// TIA Portal V19 export
FUNCTION "A0303_Sollevamento_CALL" : Void   // FC148, LAD
// stored: SetENOAutomatically false
BEGIN

REGION Network 1: <<< LATO TESTA >>>
END_REGION

REGION Network 2: Data In - Ax
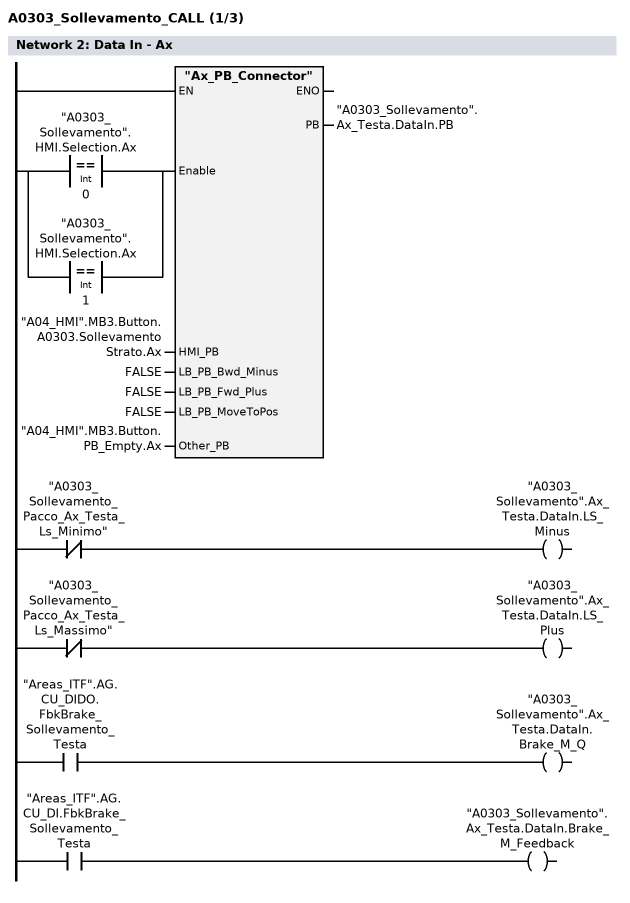
   RUNG wire#powerrail
      "Ax_PB_Connector"(Enable := wire#w1, HMI_PB := "A04_HMI".MB3.Button.A0303.SollevamentoStrato.Ax, LB_PB_Bwd_Minus := FALSE, LB_PB_Fwd_Plus := FALSE, LB_PB_MoveToPos := FALSE, Other_PB := "A04_HMI".MB3.Button.PB_Empty.Ax, PB => "A0303_Sollevamento".Ax_Testa.DataIn.PB)
   END_RUNG
   RUNG wire#powerrail
      { S7_Templates := "SrcType := Int" } EQ_Contact(in1 := "A0303_Sollevamento".HMI.Selection.Ax, in2 := 0)
   END_RUNG wire#w1
   RUNG wire#powerrail
      { S7_Templates := "SrcType := Int" } EQ_Contact(in1 := "A0303_Sollevamento".HMI.Selection.Ax, in2 := 1)
   END_RUNG wire#w1
   RUNG wire#powerrail
      I_Contact( "A0303_Sollevamento_Pacco_Ax_Testa_Ls_Minimo" )
      Coil( "A0303_Sollevamento".Ax_Testa.DataIn.LS_Minus )
   END_RUNG
   RUNG wire#powerrail
      I_Contact( "A0303_Sollevamento_Pacco_Ax_Testa_Ls_Massimo" )
      Coil( "A0303_Sollevamento".Ax_Testa.DataIn.LS_Plus )
   END_RUNG
   RUNG wire#powerrail
      Contact( "Areas_ITF".AG.CU_DIDO.FbkBrake_Sollevamento_Testa )
      Coil( "A0303_Sollevamento".Ax_Testa.DataIn.Brake_M_Q )
   END_RUNG
   RUNG wire#powerrail
      Contact( "Areas_ITF".AG.CU_DI.FbkBrake_Sollevamento_Testa )
      Coil( "A0303_Sollevamento".Ax_Testa.DataIn.Brake_M_Feedback )
   END_RUNG
   // the same network as SCL:
   "Ax_PB_Connector"(Enable := ("A0303_Sollevamento".HMI.Selection.Ax = 0) OR ("A0303_Sollevamento".HMI.Selection.Ax = 1),
                     HMI_PB := "A04_HMI".MB3.Button.A0303.SollevamentoStrato.Ax,
                     LB_PB_Bwd_Minus := FALSE,
                     LB_PB_Fwd_Plus := FALSE,
                     LB_PB_MoveToPos := FALSE,
                     Other_PB := "A04_HMI".MB3.Button.PB_Empty.Ax,
                     PB => "A0303_Sollevamento".Ax_Testa.DataIn.PB);
   "A0303_Sollevamento".Ax_Testa.DataIn.LS_Minus := NOT "A0303_Sollevamento_Pacco_Ax_Testa_Ls_Minimo";
   "A0303_Sollevamento".Ax_Testa.DataIn.LS_Plus := NOT "A0303_Sollevamento_Pacco_Ax_Testa_Ls_Massimo";
   "A0303_Sollevamento".Ax_Testa.DataIn.Brake_M_Q := "Areas_ITF".AG.CU_DIDO.FbkBrake_Sollevamento_Testa;
   "A0303_Sollevamento".Ax_Testa.DataIn.Brake_M_Feedback := "Areas_ITF".AG.CU_DI.FbkBrake_Sollevamento_Testa;
END_REGION

REGION Network 3: <<< LATO CODA >>>
END_REGION

REGION Network 4: Data In - Ax
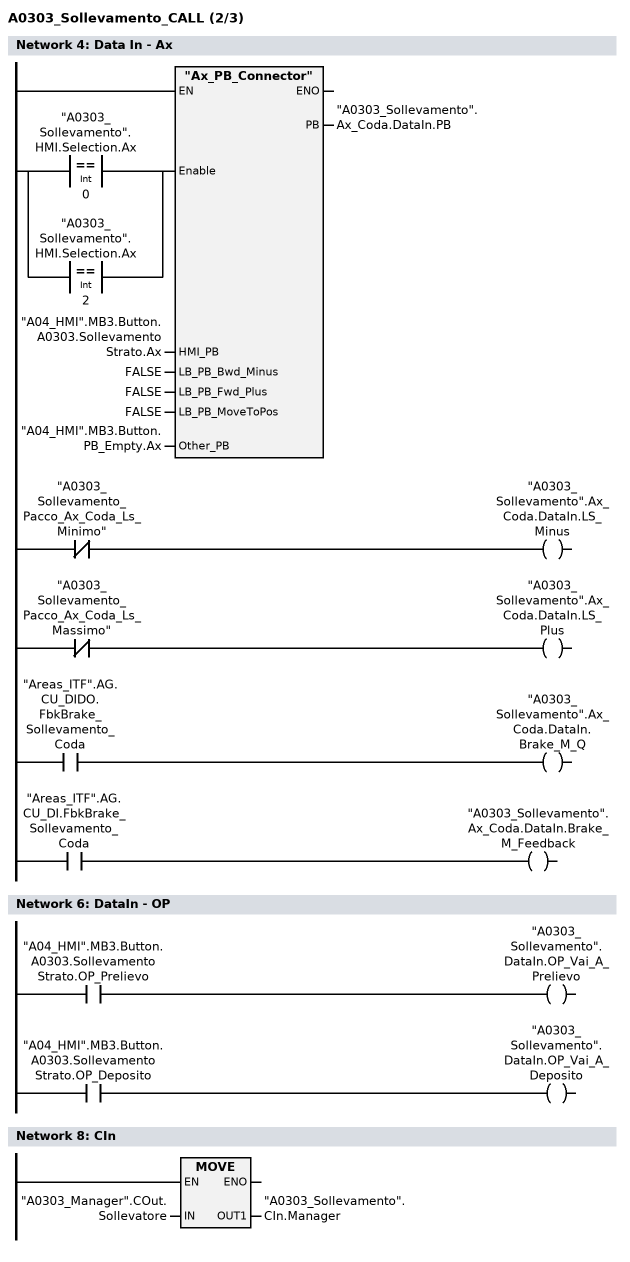
   RUNG wire#powerrail
      "Ax_PB_Connector"(Enable := wire#w1, HMI_PB := "A04_HMI".MB3.Button.A0303.SollevamentoStrato.Ax, LB_PB_Bwd_Minus := FALSE, LB_PB_Fwd_Plus := FALSE, LB_PB_MoveToPos := FALSE, Other_PB := "A04_HMI".MB3.Button.PB_Empty.Ax, PB => "A0303_Sollevamento".Ax_Coda.DataIn.PB)
   END_RUNG
   RUNG wire#powerrail
      { S7_Templates := "SrcType := Int" } EQ_Contact(in1 := "A0303_Sollevamento".HMI.Selection.Ax, in2 := 0)
   END_RUNG wire#w1
   RUNG wire#powerrail
      { S7_Templates := "SrcType := Int" } EQ_Contact(in1 := "A0303_Sollevamento".HMI.Selection.Ax, in2 := 2)
   END_RUNG wire#w1
   RUNG wire#powerrail
      I_Contact( "A0303_Sollevamento_Pacco_Ax_Coda_Ls_Minimo" )
      Coil( "A0303_Sollevamento".Ax_Coda.DataIn.LS_Minus )
   END_RUNG
   RUNG wire#powerrail
      I_Contact( "A0303_Sollevamento_Pacco_Ax_Coda_Ls_Massimo" )
      Coil( "A0303_Sollevamento".Ax_Coda.DataIn.LS_Plus )
   END_RUNG
   RUNG wire#powerrail
      Contact( "Areas_ITF".AG.CU_DIDO.FbkBrake_Sollevamento_Coda )
      Coil( "A0303_Sollevamento".Ax_Coda.DataIn.Brake_M_Q )
   END_RUNG
   RUNG wire#powerrail
      Contact( "Areas_ITF".AG.CU_DI.FbkBrake_Sollevamento_Coda )
      Coil( "A0303_Sollevamento".Ax_Coda.DataIn.Brake_M_Feedback )
   END_RUNG
   // the same network as SCL:
   "Ax_PB_Connector"(Enable := ("A0303_Sollevamento".HMI.Selection.Ax = 0) OR ("A0303_Sollevamento".HMI.Selection.Ax = 2),
                     HMI_PB := "A04_HMI".MB3.Button.A0303.SollevamentoStrato.Ax,
                     LB_PB_Bwd_Minus := FALSE,
                     LB_PB_Fwd_Plus := FALSE,
                     LB_PB_MoveToPos := FALSE,
                     Other_PB := "A04_HMI".MB3.Button.PB_Empty.Ax,
                     PB => "A0303_Sollevamento".Ax_Coda.DataIn.PB);
   "A0303_Sollevamento".Ax_Coda.DataIn.LS_Minus := NOT "A0303_Sollevamento_Pacco_Ax_Coda_Ls_Minimo";
   "A0303_Sollevamento".Ax_Coda.DataIn.LS_Plus := NOT "A0303_Sollevamento_Pacco_Ax_Coda_Ls_Massimo";
   "A0303_Sollevamento".Ax_Coda.DataIn.Brake_M_Q := "Areas_ITF".AG.CU_DIDO.FbkBrake_Sollevamento_Coda;
   "A0303_Sollevamento".Ax_Coda.DataIn.Brake_M_Feedback := "Areas_ITF".AG.CU_DI.FbkBrake_Sollevamento_Coda;
END_REGION

REGION Network 5: >
END_REGION

REGION Network 6: DataIn - OP
   RUNG wire#powerrail
      Contact( "A04_HMI".MB3.Button.A0303.SollevamentoStrato.OP_Prelievo )
      Coil( "A0303_Sollevamento".DataIn.OP_Vai_A_Prelievo )
   END_RUNG
   RUNG wire#powerrail
      Contact( "A04_HMI".MB3.Button.A0303.SollevamentoStrato.OP_Deposito )
      Coil( "A0303_Sollevamento".DataIn.OP_Vai_A_Deposito )
   END_RUNG
   // the same network as SCL:
   "A0303_Sollevamento".DataIn.OP_Vai_A_Prelievo := "A04_HMI".MB3.Button.A0303.SollevamentoStrato.OP_Prelievo;
   "A0303_Sollevamento".DataIn.OP_Vai_A_Deposito := "A04_HMI".MB3.Button.A0303.SollevamentoStrato.OP_Deposito;
END_REGION

REGION Network 7: >
END_REGION

REGION Network 8: CIn
   RUNG wire#powerrail
      Move(in := "A0303_Manager".COut.Sollevatore, out1 => "A0303_Sollevamento".CIn.Manager)
   END_RUNG
   // the same network as SCL:
   "A0303_Sollevamento".CIn.Manager := "A0303_Manager".COut.Sollevatore;
END_REGION

REGION Network 9: CIn Trasporto
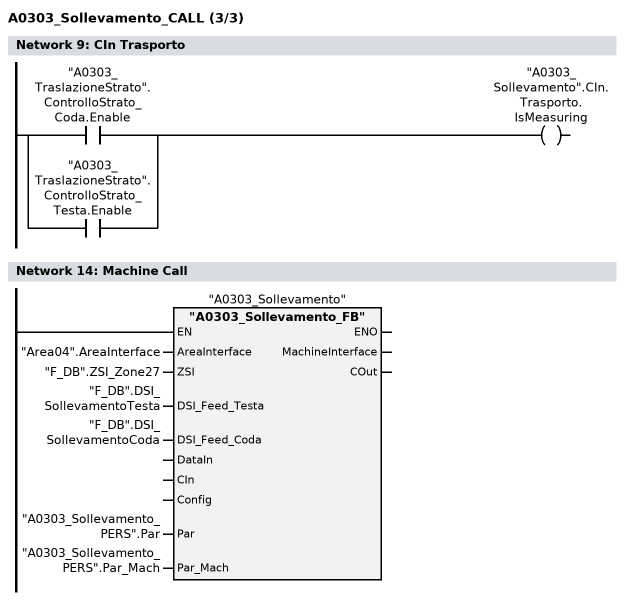
   RUNG wire#powerrail
      Contact( "A0303_TraslazioneStrato".ControlloStrato_Coda.Enable )
      wire#w1
      Coil( "A0303_Sollevamento".CIn.Trasporto.IsMeasuring )
   END_RUNG
   RUNG wire#powerrail
      Contact( "A0303_TraslazioneStrato".ControlloStrato_Testa.Enable )
   END_RUNG wire#w1
   // the same network as SCL:
   "A0303_Sollevamento".CIn.Trasporto.IsMeasuring := "A0303_TraslazioneStrato".ControlloStrato_Coda.Enable OR "A0303_TraslazioneStrato".ControlloStrato_Testa.Enable;
END_REGION

REGION Network 10: >
END_REGION

REGION Network 11 (SCL): Drive
   "A0303_Sollevamento".Ax_Testa.Drive.Infeed_ON := "Areas_ITF".AG.Infeed_Running;
   "A0303_Sollevamento".Ax_Testa.Drive.AccessPoint := "HW_Const_Values".CU8_PN_615A1_ModuleAccessPoint;
   "A0303_Sollevamento".Ax_Testa.Drive.AxisID := "CU8_ID_2_2390A1_1_2390M1";
   "A0303_Sollevamento".Ax_Testa.Drive.TokenChain := "TOKENCHAIN_CU8";

   "A0303_Sollevamento".Ax_Coda.Drive.Infeed_ON := "Areas_ITF".AG.Infeed_Running;
   "A0303_Sollevamento".Ax_Coda.Drive.AccessPoint := "HW_Const_Values".CU8_PN_615A1_ModuleAccessPoint;
   "A0303_Sollevamento".Ax_Coda.Drive.AxisID := "CU8_ID_3_2390A1_2_2400M1";
   "A0303_Sollevamento".Ax_Coda.Drive.TokenChain :=  "TOKENCHAIN_CU8";
END_REGION

REGION Network 12 (SCL): HW ID
   "A0303_Sollevamento".Ax_Testa.HW_ID_TEL1 := "HW_Const_Values".CU8_PN_2390A1_1_Standard_telegram_1;
   "A0303_Sollevamento".Enc_Testa.HW_IO := "HW_Const_Values".HW_2394P1_Telegram_81_DI_DO;

   "A0303_Sollevamento".Ax_Coda.HW_ID_TEL1 := "HW_Const_Values".CU8_PN_2390A1_2_Standard_telegram_1;
   "A0303_Sollevamento".Enc_Coda.HW_IO := "HW_Const_Values".HW_2404P1_Telegram_81_DI_DO;
END_REGION

REGION Network 13: >
END_REGION

REGION Network 14: Machine Call
   RUNG wire#powerrail
      "A0303_Sollevamento"(AreaInterface := "Area04".AreaInterface, ZSI := "F_DB".ZSI_Zone27, DSI_Feed_Testa := "F_DB".DSI_SollevamentoTesta, DSI_Feed_Coda := "F_DB".DSI_SollevamentoCoda, DataIn :=, CIn :=, Config :=, Par := "A0303_Sollevamento_PERS".Par, Par_Mach := "A0303_Sollevamento_PERS".Par_Mach, MachineInterface =>, COut =>)
   END_RUNG
   // the same network as SCL:
   "A0303_Sollevamento"(AreaInterface := "Area04".AreaInterface,   // "A0303_Sollevamento_FB"
                        ZSI := "F_DB".ZSI_Zone27,
                        DSI_Feed_Testa := "F_DB".DSI_SollevamentoTesta,
                        DSI_Feed_Coda := "F_DB".DSI_SollevamentoCoda,
                        Par := "A0303_Sollevamento_PERS".Par,
                        Par_Mach := "A0303_Sollevamento_PERS".Par_Mach);
END_REGION

REGION Network 15: >
END_REGION

REGION Network 16: >
END_REGION

REGION Network 17: >
END_REGION
END_FUNCTION
